(*********************************** G.D S.p.A. - Technical Department ***********************************
============= PROGRAM INFO ============
FOLDER:             TBD
MACHINES INVOLVED:  TBD 

============= DESCRIPTION =============
csp machine declaration

============= REVISIONS ===============
Date		Version	 	Author      	Description             
----------	-------		------------  	--------------------------------------------
2019/04/05 	0000.00	 	M.Grasso		Creation of the PRG

**********************************************************************************************************)
(*$R process_ref := prc; $*)
PROGRAM csp_transfer_infeed_accU
VAR
	
	prc:											process;
	prc_path:										STRING;
	
END_VAR

_read_var_input();

_object_manager();

IF NOT objects_running()
THEN
	RETURN;	
END_IF

_read_process_image();

_mode_manager();

_set_runtime_properties();

(********************************* BODY *********************************)
(************************************************************************)

_handle_messages();

_write_output();

ACTION _handle_messages:
;
END_ACTION

ACTION _handle_process_test:
;
END_ACTION

ACTION _mode_manager:
IF process_mode_req_is_pending(prc)
THEN
    process_apply_mode_req_first_step(prc);
    CASE process_get_mode(prc) OF
        MODE_TO_ABSENT:
			;
        MODE_TO_INACTIVE:
			;
        MODE_TO_TEST:
			;
        MODE_TO_OPERATIONAL:
			;
    END_CASE
    process_apply_mode_req_second_step(prc);
END_IF
END_ACTION

ACTION _object_manager:
IF objects_initialization()
THEN
	sub_process_init(
		object_name					:= 'csp_transfer_infeed_accU.prc', 
		process						:= csp_transfer_infeed.prc, 
		CONVERSION_this				:= prc);
		
	prc_path 						:= process_get_path(prc);
END_IF

IF objects_running()
THEN
	process_cycle(prc);
END_IF
END_ACTION

ACTION _read_process_image:
;
END_ACTION

ACTION _read_var_input:
;
END_ACTION

ACTION _set_runtime_properties:
;
END_ACTION

ACTION _write_output:
;
END_ACTION

END_PROGRAM

(* stored: Version 1.1.0.1, ProductVersion 3.1.4022.12
   POU csp_transfer_infeed_accU: Id {3602caae-4837-4882-a3ea-4593b97c30fb}, SpecialFunc None
   Action _handle_messages: Id {2f304be9-5ef2-44e2-83ee-93bf0ba7c1a2}
   Action _handle_process_test: Id {9e1ba91f-7dfe-469a-8a7e-a7739f7cb38e}
   Action _mode_manager: Id {ee3fdb79-97fd-4534-b4c4-7aa54e016e28}
   Action _object_manager: Id {e66ed7f0-c1d5-4607-8e84-0ae1992a6af3}
   Action _read_process_image: Id {a93ad75f-0f27-4fc8-bb80-5329d67d13d6}
   Action _read_var_input: Id {c239819a-c279-4259-b7ab-cc0a6ea2319d}
   Action _set_runtime_properties: Id {7fc970e0-c014-4c3e-9d95-cab064a6fb3c}
   Action _write_output: Id {2d0d7e32-e9d4-4499-9d8a-548f5993de3b} *)
